FUNCTION_BLOCK Executer_Object EXTENDS TcoCore.TcoObject
VAR
END_VAR

{attribute 'hide'}
PROPERTY Identity : ULINT
GET
Identity := 0;
END_GET
END_PROPERTY

END_FUNCTION_BLOCK

(* stored: Version 1.1.0.1, ProductVersion 3.1.4024.6
   POU Executer_Object: Id {6cf2ba54-d2cb-0a9f-316a-a860ff9dc167}, SpecialFunc None
   Property Identity: Id {95bef5fa-169e-0173-37b9-b1fdfef23db6}
   Get Get: Id {3212a690-c280-0ebe-1ded-a4e9a2b594c5} *)
